FUNCTION_BLOCK ApplicationManager EXTENDS PAClassAlarmingBase
VAR_INPUT
END_VAR
VAR_OUTPUT
END_VAR
VAR
END_VAR

END_FUNCTION_BLOCK

(* stored: Version 1.1.0.1, ProductVersion 3.1.4020.12
   POU ApplicationManager: Id {b0d12743-9b42-4cee-8ff9-bcbf4e85167d}, SpecialFunc None *)
